{attribute 'no_explicit_call' := 'This FB is a CLASS and must be accessed using methods or properties'}
{attribute 'enable_dynamic_creation'}
//{attribute 'hide_all_locals'}
FUNCTION_BLOCK FB_DynamicArrayOfLREAL
VAR
	buffer : FB_JsonDomParser;
	root : sJsonValue;
END_VAR

PROPERTY PRIVATE _Array : sJsonValue
GET
IF root <> 0 THEN
	_Array := root;
ELSE
	root := buffer.NewDocument();
	_Array := buffer.SetArray(root,0);
END_IF
END_GET
END_PROPERTY

METHOD PUBLIC AddLast : BOOL
VAR_IN_OUT
	Value : LREAL;
END_VAR
AddLast := buffer.PushbackDoubleValue(v:= _Array, Value) <> 0;
END_METHOD

METHOD PUBLIC Clear : BOOL
VAR
	_arrayElement : SJsonAIterator;
END_VAR
_arrayElement := buffer.ArrayBegin(_array);
IF _arrayElement <> 0 THEN
	Clear := buffer.ClearArray(v := _array,i := _arrayElement);
END_IF
END_METHOD

METHOD PUBLIC CopyArrayString : BOOL
VAR_IN_OUT CONSTANT
  	pDoc : STRING; 
END_VAR
VAR_INPUT
	nDoc : UDINT;
END_VAR
CopyArrayString := buffer.copyjson(v:= _Array, pDoc:= pDoc,nDoc := nDoc) <> 0;
END_METHOD

PROPERTY PUBLIC Count : UDINT
GET
Count := buffer.GetArraySize(_array);
END_GET
END_PROPERTY

PROPERTY PUBLIC FirstIndex : UDINT
GET
FirstIndex := 0;
END_GET
END_PROPERTY

PROPERTY PUBLIC LastIndex : UDINT
GET
IF Count = 0 THEN
	LastIndex := 0;
ELSE 
	LastIndex := Count - 1;
END_IF
END_GET
END_PROPERTY

METHOD PUBLIC RemoveFirst : BOOL
VAR
	_arrayElement : SJsonAIterator;
END_VAR
RemoveFirst := TryDeleteIndex(0);
END_METHOD

METHOD PUBLIC RemoveLast: BOOL
VAR
	_arrayElement : SJsonAIterator;
END_VAR
RemoveLast := TryDeleteIndex(LastIndex);
END_METHOD

METHOD PUBLIC TryDeleteIndex : BOOL
VAR_INPUT
	Index : UDINT;
END_VAR
VAR
	_arrayElement : SJsonAIterator;
END_VAR
_arrayElement := buffer.GetArrayValueByIdx(_Array, Index);
IF _arrayElement <> 0 THEN
	TryDeleteIndex := buffer.RemoveArray(v := _array,i := _arrayElement);
END_IF
END_METHOD

METHOD PUBLIC TryGetIndex : BOOL;
VAR_INPUT
	Index : UDINT;	
END_VAR
VAR_IN_OUT
	Destination : LREAL;
END_VAR
Destination := buffer.GetDouble(v:= buffer.GetArrayValueByIdx(_Array, Index));
END_METHOD

METHOD PUBLIC TrySetIndex : BOOL
VAR_INPUT
	Index : UDINT;
END_VAR
VAR_IN_OUT
	Value : LREAL;
END_VAR
TrySetIndex := buffer.SetDouble(v:= buffer.GetArrayValueByIdx(_Array, Index),Value) <> 0;
END_METHOD

END_FUNCTION_BLOCK

(* stored: Version 1.1.0.1, ProductVersion 3.1.4024.12
   POU FB_DynamicArrayOfLREAL: Id {ebf24724-4612-46a8-8cdc-f13249909af4}, SpecialFunc None
   Folder Private: Id {7a72a895-9b7e-4075-85b1-8890248cc693}
   Property _Array: Id {3788a386-b8a0-4ddc-9e99-5ddc70f1e40f}
   Get Get: Id {7fc147fd-6548-4819-80b0-4c2516beed43}
   Method AddLast: Id {31713e8f-7edc-49a3-8ffb-b5d5bea623c8}
   Method Clear: Id {ec35813b-0062-4622-b687-ac935f36693d}
   Method CopyArrayString: Id {839fb1de-1c7c-49ea-908b-124851825a53}
   Property Count: Id {624efaf4-940a-411a-ba0b-ea6fcbb425a0}
   Get Get: Id {321bb1c8-2534-41b6-936f-8104ce1b4687}
   Property FirstIndex: Id {434da13a-ffc8-4709-ab33-6efab001ef45}
   Get Get: Id {535a91e8-9138-4fe4-858c-4604c33bd049}
   Property LastIndex: Id {7d873392-e487-4475-b90f-0976c401e968}
   Get Get: Id {bf529785-d9e0-444d-9101-ab47546a8281}
   Method RemoveFirst: Id {71b667b0-e59c-44b7-815c-159f05453e17}
   Method RemoveLast: Id {86669941-2f8b-4969-857d-96623596bd6f}
   Method TryDeleteIndex: Id {ff975f21-3e61-4ecc-b5fb-cb6a42c35c34}
   Method TryGetIndex: Id {72daf367-4658-458b-bfae-b5724022a5ff}
   Method TrySetIndex: Id {0baf6dfb-f78c-443c-926b-7af1af08e01f} *)
